TYPE "PLCtoMES_ResultsStoredScanExchange_ext"
VERSION : 0.1
   STRUCT
      Load_Scanner1ChickInReq : Bool;
      Load_Scanner2ChickInReq : Bool;
      Load_Scanner3ChickInReq : Bool;
      Load_Scanner4ChickInReq : Bool;
      Load_Scanner5ChickInReq : Bool;
      Load_Scanner6ChickInReq : Bool;
      Load_Scanner7ChickInReq : Bool;
      Load_Scanner8ChickInReq : Bool;
      SpareByte : Byte;
   END_STRUCT;

END_TYPE

